DATA_BLOCK "MotorContro_DB_16"
{ S7_Optimized_Access := 'TRUE' }
VERSION : 0.1
NON_RETAIN
"MotorContro"

BEGIN

END_DATA_BLOCK

